{attribute 'GeneratedUsingTerminal: EK1122-0000-0018'}
{attribute addProperty BoxType "EK1122-0000-0018"}
{attribute addProperty Id "Beckhoff_EL67xxsub_EK1100EK1100_1FC0878B2"}
{attribute addProperty CRC "1213625614"}
{attribute addProperty Size "2"}
TYPE Beckhoff_EL67xxEK1122_4856750E EXTENDS EK1122_1FC0878B :
STRUCT
	{attribute addProperty Name "Beckhoff_EL67xxsub_EK1100"}
	{attribute addProperty PreviousPort "Beckhoff EL67xxEK1122 : D"}
	Beckhoff_EL67xxsub_EK1100 : EK1100_1FC0878B;
END_STRUCT
END_TYPE

(* stored: Version 1.2.0.0, ProductVersion 3.1.4024.9
   DUT Beckhoff_EL67xxEK1122_4856750E: Id {4409e813-6821-438c-aab8-37298f517fd5} *)
